D36187	WORD	OK/NG마스타 G8:RR LH "T" REAL Data 차이 <RG3 EV>
D36190	WORD	W500 G9:RR LH "L" REAL Data 차이 <RG3 EV>
D36192	WORD	OK/NG마스타 G9:RR LH "L" REAL Data 차이 <RG3 EV>
D36195	WORD	W500 G10:RR LH "H" REAL Data 차이 <RG3 EV>
D36197	WORD	OK/NG마스타 G10:RR LH "H" REAL Data 차이 <RG3 EV>
D36200	WORD	W500 G11:RR RH "T" REAL Data 차이 <RG3 EV>
D36202	WORD	OK/NG마스타 G11:RR RH "T" REAL Data 차이 <RG3 EV>
D36205	WORD	W500 G12:RR RH "L" REAL Data 차이 <RG3 EV>
D36207	WORD	OK/NG마스타 G12:RR RH "L" REAL Data 차이 <RG3 EV>
D36210	WORD	W500 G13:RR RH "H" REAL Data 차이 <RG3 EV>
D36212	WORD	OK/NG마스타 G13:RR RH "H" REAL Data 차이 <RG3 EV>
D36250	WORD	W600 G1:CTR "L" REAL Data 차이 <RG3 EV>
D36255	WORD	W600 G2:FRT LH "T" REAL Data 차이 <RG3 EV>
D36260	WORD	W600 G3:FRT LH "L" REAL Data 차이 <RG3 EV>
D36265	WORD	W600 G4:FRT LH "H" REAL Data 차이 <RG3 EV>
D36270	WORD	W600 G5:FRT RH "T" REAL Data 차이 <RG3 EV>
D36275	WORD	W600 G6:FRT RH "L" REAL Data 차이 <RG3 EV>
D36280	WORD	W600 G7:FRT RH "H" REAL Data 차이 <RG3 EV>
D36285	WORD	W600 G8:RR LH "T" REAL Data 차이 <RG3 EV>
D36290	WORD	W600 G9:RR LH "L" REAL Data 차이 <RG3 EV>
D36295	WORD	W600 G10:RR LH "H" REAL Data 차이 <RG3 EV>
D36300	WORD	W600 G11:RR RH "T" REAL Data 차이 <RG3 EV>
D36305	WORD	W600 G12:RR RH "L" REAL Data 차이 <RG3 EV>
D36310	WORD	W600 G13:RR RH "H" REAL Data 차이 <RG3 EV>
K01892	BIT	비젼 마스타 기동 W300 배출
D27040	WORD	W350 스케너 Data_LH (W400)
D27540	WORD	W350 스케너 Data_RH (W400)
D27060	WORD	W350 스케너 Data_LH (W400 -> HD2)
D27560	WORD	W350 스케너 Data_RH (W400 -> HD2)
D27080	WORD	W350 스케너 Data_LH (HD2 -> W500)
D27580	WORD	W350 스케너 Data_RH (HD2 -> W500)
D29000	WORD	W500 동도 측정 DATA 아스키 (W500 -> HD2)
D01860	WORD	W500 동도 판정 (HD2 -> W600)
D01960	WORD	W350 3D비젼 체크 (HD2 -> W600)
D24800	WORD	W500 동도 측정 DATA 실수 (HD2 -> NG 대차)
D27160	WORD	W350 스케너 Data_LH (HD2 -> NG 대차)
D27660	WORD	W350 스케너 Data_RH (HD2 -> NG 대차)
D30000	WORD	W500 동도 판정 (HD2 -> W700)
D32000	WORD	W500 동도 측정 DATA 실수 (HD2 -> W700)
D27180	WORD	W350 스케너 Data_LH (HD2 -> W700)
D27680	WORD	W350 스케너 Data_RH (HD2 -> W700)
D30030	WORD	W500 동도 판정 (W700 -> HD2)
D32200	WORD	W500 동도 측정 DATA 실수 (W700 -> HD2)
D33800	WORD	W500 동도 측정 DATA 아스키 (W700 -> HD2)
D30060	WORD	W500 동도 판정 (HD2 -> PLT)
D32400	WORD	W500 동도 측정 DATA 실수 (HD2 -> PLT)
D34000	WORD	W500 동도 측정 DATA 아스키 (HD2 -> PLT)
D27200	WORD	W350 스케너 Data_LH (W700 -> HD2)
D27220	WORD	W350 스케너 Data_LH (HD2 -> PLT)
D27700	WORD	W350 스케너 Data_RH (W700 -> HD2)
D27720	WORD	W350 스케너 Data_RH (HD2 -> PLT)
P0050C	BIT	W10 RH 1차 클램프 잠김1
P0050E	BIT	W10 RH 1차 클램프 잠김2
M10821	BIT	R08 HD2 (In18) PLT-A PLT 사양 확인 
M10824	BIT	R08 HD2 (In21) PLT-B PLT 사양 확인 
K00003	BIT	차종.3 RS4
M10712	BIT	R07 HD1 (In03) 차종3
M10713	BIT	R07 HD1 (In04) 차종4
M10714	BIT	R07 HD1 (In05) 차종5
M10715	BIT	R07 HD1 (In06) 차종6
M10716	BIT	R07 HD1 (In07) 차종7
M10717	BIT	R07 HD1 (In08) 차종8
M10812	BIT	R08 HD2 (In03) 차종3
M10813	BIT	R08 HD2 (In04) 차종4
M10814	BIT	R08 HD2 (In05) 차종5
M10815	BIT	R08 HD2 (In06) 차종6
M10816	BIT	R08 HD2 (In07) 차종7
M10817	BIT	R08 HD2 (In08) 차종8
T0217	BIT/WORD	W10 RH 사양감지 체크완료 지연
M01006	BIT	W250 서보 동작가능
M0100B	BIT	W250 상부 안전센서 정상
M0100C	BIT	W250 하부 안전세서 정상
M0100D	BIT	W250 안전매트 정상
M01060	BIT	W250 원위치복귀 Pb (XP)
M01074	BIT	W250 4차 기동
T1003	BIT/WORD	W250 Air Blow On TMR
T1016	BIT/WORD	W250 파트이상 (누락)지연
T1018	BIT/WORD	W250 서보 위치이상 지연
T1019	BIT/WORD	W250 서보 근접센서 위치이상 Tmr
P0241C	BIT	W70 기동-L
P0241D	BIT	W70 기동-R
P0241E	BIT	W70 원점복귀
D06230	WORD	Label Text.6 Count Data
D00065	WORD	Barcode QR Code Count Data
D00060	WORD	Label Count
D06200	WORD	Label "Year"
D06202	WORD	Label "Month"
D06203	WORD	Label "Day"
D00067	WORD	Barcode QR Code Count ReData
D06210	WORD	Label QR Code Count
D06236	WORD	Label TEXT.6 Count ReData
D06220	WORD	Label TEXT.6 Count Send
D21050	WORD	Label QR Code "0,6,GS,V"
D21054	WORD	Label QR Code "GS,P"
D21060	WORD	Label QR Code "GS,S"
D21068	WORD	Label QR Code "GS,T"
D06201	WORD	Label Year, Month, Day
D21069	WORD	Label QR Code Date Year,Month,Day Send
D21074	WORD	Label QR Code (A0) Send
D21075	WORD	Label QR Code Count Send
D05900	WORD	Lable QR Code Worker Data
D21090	WORD	Label Text.6 Count Send
D20500	WORD	Label QR Code ([)>RS) Send
D20540	WORD	Label Text.5 Date Send
D20541	WORD	Label Text.5 Date Send
D20542	WORD	Label Text.5 Date Send
D20543	WORD	Label Text.5 Date Send
D20544	WORD	Label Text.5 Date Send
D20550	WORD	Label QR Code "0,6,GS,V"
D20554	WORD	Label QR Code "GS,P"
D20560	WORD	Label QR Code "GS,S"
D20563	WORD	Label le QR Code "GS,E"
D20568	WORD	Label QR Code "GS,T"
D20569	WORD	Label QR Code Date Year,Month,Day Send
D20573	WORD	Label QR Code Worker Data
D20574	WORD	Label QR Code (A0) Send
D20575	WORD	Label QR Code Count Send
D20590	WORD	Label Text.6 Count Send
D20541.0	BIT	/
D20541.8	BIT	Label "Month1"
D20542.0	BIT	Label "Month2"
D20542.8	BIT	/
D00099.0	BIT	Label Manual Print
M08511	BIT	ZEBRA Label Head Send
M08512	BIT	ZEBRA Text1 Position Send
M08513	BIT	ZEBRA Text2 Position Send 
M08521	BIT	ZEBRA Text1 Data Send
M08522	BIT	ZEBRA Text2 Data Send
M08523	BIT	ZEBRA Text3 Data Send
M08514	BIT	ZEBRA Text3 Position Send
M08515	BIT	ZEBRA Text4 Position Send
M08524	BIT	ZEBRA Text4 Data Send
M08525	BIT	ZEBRA Text5 Data Send
M08516	BIT	ZEBRA Text5 Position Send
M08517	BIT	ZEBRA Text6 Position Send
M08526	BIT	ZEBRA Text6 Data Send
M08518	BIT	ZEBRA 2D Code Position Send
M08527	BIT	ZEBRA 2D Code Data Send
M08550	BIT	Label Print Complete
P02417	BIT	W70 공기압력
P0241A	BIT	W70 광 안전장치_상부1
P0241B	BIT	W70 광 안전장치_상부2
P02400	BIT	W70 클램프 전진1
P02402	BIT	W70 클램프 전진2
P02404	BIT	W70 클램프 전진3
P02406	BIT	W70 클램프 전진4
P02401	BIT	W70 클램프 후진1
P02403	BIT	W70 클램프 후진2
P02405	BIT	W70 클램프 후진3
P02407	BIT	W70 클램프 후진4
P02408	BIT	W70 동도 유니트 상승1
P0240A	BIT	W70 동도 유니트 상승2
P0240C	BIT	W70 동도 유니트 상승3
P02409	BIT	W70 동도 유니트 하강1
P0240B	BIT	W70 동도 유니트 하강2
P0240D	BIT	W70 동도 유니트 하강3
P02410	BIT	W70 제품확인1
P02411	BIT	W70 제품확인2
P02420	BIT	W70 클램프 잠김 Sol
P02421	BIT	W70 클램프 풀림 Sol
P02422	BIT	W70 동도 유니트 상승 Sol
P02423	BIT	W70 동도 유니트 하강 Sol
P02440	BIT	[From] W500 TOE/CAM Ready
P02441	BIT	[From] W500 TOE/CAM ERROR
P02442	BIT	[From] W500 TOE/CAM N.G
P02443	BIT	[From] W500 TOE/CAM O.K
P02450	BIT	[To Dongdo] W500TOE/CAM Model1
P02451	BIT	[To Dongdo] W500TOE/CAM Model2
P02452	BIT	[To Dongdo] W500TOE/CAM Model4
P02453	BIT	[To Dongdo] W500TOE/CAM Model8
P02454	BIT	[To Dongdo] W500 TOE/CAM Check Start
D41000	WORD	W70 동도 버퍼
D44000	WORD	W70 동도 측정 DATA
D41003	WORD	P1 ASCII Data
D41008	WORD	P2 ASCII Data
D41013	WORD	P3 ASCII Data
D41018	WORD	P4 ASCII Data
D41023	WORD	P5 ASCII Data
D41028	WORD	P6 ASCII Data
D41033	WORD	P7 ASCII Data
D42000	WORD	동도 읽을 위치 1
D42001	WORD	동도 읽을 자릿수 1
D42002	WORD	동도 읽을 위치 2
D42003	WORD	동도 읽을 자릿수 2
D42010	WORD	P1 ASCII Data
D42020	WORD	P2 ASCII Data
D42030	WORD	P3 ASCII Data
D42040	WORD	P4 ASCII Data
D42050	WORD	P5 ASCII Data
D42060	WORD	P6 ASCII Data
D42070	WORD	P7 ASCII Data
D44010	WORD	P1 REAL Data
D44020	WORD	P2 REAL Data
D44030	WORD	P3 REAL Data
D44040	WORD	P4 REAL Data
D44050	WORD	P5 REAL Data
D44060	WORD	P6 REAL Data
D44070	WORD	P7 REAL Data
D45007	WORD	Data 절대 상/하한치
D45010	WORD	P1 REAL Data 하한치
D45012	WORD	P1 REAL Data 하한치 절대
D45015	WORD	P1 REAL Data 상한치
D45017	WORD	P1 REAL Data 상한치 절대
D45020	WORD	P2 REAL Data 하한치
D45022	WORD	P2 REAL Data 하한치 절대
D45025	WORD	P2 REAL Data 상한치
D45027	WORD	P2 REAL Data 상한치 절대
D45030	WORD	P3 REAL Data 하한치
D45032	WORD	P3 REAL Data 하한치 절대
D45035	WORD	P3 REAL Data 상한치
D45037	WORD	P3 REAL Data 상한치 절대
D45040	WORD	P4 REAL Data 하한치
D45042	WORD	P4 REAL Data 하한치 절대
D45045	WORD	P4 REAL Data 상한치
D45047	WORD	P4 REAL Data 상한치 절대
D45050	WORD	P5 REAL Data 하한치
D45052	WORD	P5 REAL Data 하한치 절대
D45055	WORD	P5 REAL Data 상한치
D45057	WORD	P5 REAL Data 상한치 절대
D45060	WORD	P6 REAL Data 하한치
D45062	WORD	P6 REAL Data 하한치 절대
D45065	WORD	P6 REAL Data 상한치
D45067	WORD	P6 REAL Data 상한치 절대
D45070	WORD	P7 REAL Data 하한치
D45072	WORD	P7 REAL Data 하한치 절대
D45075	WORD	P7 REAL Data 상한치
D45077	WORD	P7 REAL Data 상한치 절대
D46010	WORD	P1 REAL 스펙Data 
D46012	WORD	P1 REAL 하한치
D46017	WORD	P1 REAL 상한치
D46020	WORD	P2 REAL 스펙Data 
D46030	WORD	P3 REAL 스펙Data 
D46040	WORD	P4 REAL 스펙Data 
D46042	WORD	P4 REAL 하한치
D46047	WORD	P4 REAL 상한치
D46050	WORD	P5 REAL 스펙Data 
D46052	WORD	P5 REAL 하한치
D46057	WORD	P5 REAL 상한치
D46060	WORD	P6 REAL 스펙Data 
D46062	WORD	P6 REAL 하한치
D46067	WORD	P6 REAL 상한치
D46070	WORD	P7 REAL 스펙Data 
D46072	WORD	P7 REAL 하한치
D46077	WORD	P7 REAL 상한치
D46150	WORD	P1 REAL Data 차이
D46155	WORD	P2 REAL Data 차이
D46160	WORD	P3 REAL Data 차이
D46165	WORD	P4 REAL Data 차이
D46170	WORD	P5 REAL Data 차이
D46175	WORD	P6 REAL Data 차이
D46180	WORD	P7 REAL Data 차이
D11007	WORD	W70 Scan Data 1
D11009	WORD	W70 Scan Data 3
D11011	WORD	W70 Scan Data 5
D31400	WORD	PLC->PC W70 스케너 Data
D31500	WORD	PLC->PC W70 동도 측정 Data
D00059.0	BIT	1 Shift Time
D00059.1	BIT	2 Shift Time
D14103.3	BIT	W70 Check OK
D14103.4	BIT	W70 Check NG
D14103.5	BIT	W70 Scan Comple
D14101.5	BIT	W70 Scan Compl
D14103.E	BIT	W70 Loading
D14101.E	BIT	W70 Loading Check
D20576	WORD	Barcord Print Data1
D15002.9	BIT	W70 수동모드
P02428	BIT	W70 타워램프-R
P02429	BIT	W70 타워램프-G
D43010	WORD	W70 P1 REAL Data_Master
D43020	WORD	W70 P2 REAL Data_Master
D43030	WORD	W70 P3 REAL Data_Master
D43040	WORD	W70 P4 REAL Data_Master
D43050	WORD	W70 P5 REAL Data_Master
D43060	WORD	W70 P6 REAL Data_Master
D43070	WORD	W70 P7 REAL Data_Master
D48150	WORD	W70 P1 REAL Data 차이 _Master
D48155	WORD	W70 P2 REAL Data 차이 _Master
D48160	WORD	W70 P3 REAL Data 차이 _Master
D48165	WORD	W70 P4 REAL Data 차이 _Master
D48170	WORD	W70 P5 REAL Data 차이 _Master
D48175	WORD	W70 P6 REAL Data 차이 _Master
D48180	WORD	W70 P7 REAL Data 차이 _Master
K01780	BIT	W70 OK 마스타 선택중
K01781	BIT	W70 OK 마스타 체크 기동
M03981	BIT	W70 OK 마스타 체크 Off T/K
M03980	BIT	W70 OK 마스타 체크 On T/K
M03984	BIT	W70 OK 마스타 예약기동
K01990	BIT	W70 OK 마스타 선택중
M05960	BIT	W70 OK 마스타 체크 On T/K
M05964	BIT	W70 OK 마스타 예약기동
K01991	BIT	W70 OK 마스타 체크 기동
M05961	BIT	W70 OK 마스타 체크 Off T/K
M05970	BIT	W70 OK 마스타 Start Lamp
R02600	WORD	W70 OK 마스타체크 최종점검 일자 년
M05971	BIT	W70 OK 마스타 주간 초품 확인시간
M05972	BIT	W70 OK 마스타 주간 중품 확인시간
M05973	BIT	W70 OK 마스타 야간 초품 확인시간
M05974	BIT	W70 OK 마스타 야간 중품 확인시간
M05951	BIT	W70 OK 마스타 주간 초품 체크 완료
M05952	BIT	W70 OK 마스타 주간 중품 체크 완료
M05953	BIT	W70 OK 마스타 야간 초품 체크 완료
M05954	BIT	W70 OK 마스타 야간 중품 체크 완료
D00029	WORD	W70 OK 마스타운영 시간설정 비번
D05822	WORD	W70 OK 마스타 주간 초품 시작 시간
D05823	WORD	W70 OK 마스타 주간 초품 끝 시간
D05824	WORD	W70 OK 마스타 주간 중품 시작 시간
D05825	WORD	W70 OK 마스타 주간 중품 끝 시간
D05826	WORD	W70 OK 마스타 야간 초품 시작 시간
D05828	WORD	W70 OK 마스타 야간 중품 시작 시간
D05827	WORD	W70 OK 마스타 야간 초품 끝 시간
D05829	WORD	W70 OK 마스타 야간 중품 끝 시간
D05840	WORD	W70 OK 마스타 주간 초품 정보
D05841	WORD	W70 OK 마스타 주간 중품 정보
D05842	WORD	W70 OK 마스타 야간 초품 정보
D05843	WORD	W70 OK 마스타 야간 중품 정보
D05820	WORD	W70 OK 마스타 확인 정보 클리어 시
D05821	WORD	W70 OK 마스타 확인 정보 클리어 분
M0597A	BIT	W70 OK마스타 주간 초품 체크 지령
M0597B	BIT	W70 OK 마스타 주간 중품 체크 지령
M0597C	BIT	W70 OK 마스타 야간 초품 체크 지령
M0597D	BIT	W70 OK 마스타 야간 중품 체크 지령
P11100	BIT	R11 HD3 Running
P11101	BIT	R11 HD3 Servo_ON
P11103	BIT	R11 HD3 Error
P11105	BIT	R11 HD3 REMOTE Mode
P11106	BIT	R11 HD3 PLAY Mode
P11107	BIT	R11 HD3 TEACH 모드
P1110A	BIT	R11 HD3 HOME Position
P11110	BIT	R11 HD3 (Ot01) W50 간섭무
P11111	BIT	R11 HD3 (Ot02) W60-1 간섭무
P11112	BIT	R11 HD3 (Ot03) W60-2 간섭무
P11113	BIT	R11 HD3 (Ot03) W60-3 간섭무
P11114	BIT	R11 HD3 (Ot05) W70 간섭무
P11115	BIT	R11 HD3 (Ot06)
P11116	BIT	R11 HD3 (Ot07)
P11117	BIT	R11 HD3 (Ot08)
P11118	BIT	R11 HD3 (Ot09) W50 언로딩 완료
P11119	BIT	R11 HD3 (Ot09)
P1111A	BIT	R11 HD3 (Ot11) W60-1 로딩 완료
P1111B	BIT	R11 HD3 (Ot12) W60-1 언로딩 완료
P1111C	BIT	R11 HD3 (Ot13) W60-2 로딩 완료
P1111D	BIT	R11 HD3 (Ot14) W60-1 언로딩 완료
P1111E	BIT	R11 HD3 (Ot15) W60-3 로딩 완료
P1111F	BIT	R11 HD3 (Ot16) W60-1 언로딩 완료
P11120	BIT	R11 HD3 (Ot17) W70 로딩완료
P11121	BIT	R11 HD3 (Ot18)
P11122	BIT	R11 HD3 (Ot19)
P11123	BIT	R11 HD3 (Ot20)
P11124	BIT	R11 HD3 (Ot21)
P11125	BIT	R11 HD3 (Ot22)
P11126	BIT	R11 HD3 (Ot23)
P11127	BIT	R11 HD3 (Ot24)
P11128	BIT	R11 HD3 (Ot25)
P11129	BIT	R11 HD3 (Ot26) R11 HD3->R01 인터록
P1112A	BIT	R11 HD3 (Ot27)
P1112B	BIT	R11 HD3 (Ot28)
P1112C	BIT	R11 HD3 (Ot29)
P1112D	BIT	R11 HD3 (Ot30)
P1112F	BIT	R11 HD3 (Ot32) 비상정지
P11131	BIT	R11 HD4 (Ot34)
P11132	BIT	R11 HD3 (Ot35)
P11133	BIT	R11 HD3 (Ot36)
P11134	BIT	R11 HD3 (Ot37)
P11135	BIT	R11 HD3 (Ot38)
P11136	BIT	R11 HD3 (Ot39)
P11137	BIT	R11 HD3 (Ot40)
P11141	BIT	R11 HD3 (Ot50) 그리퍼1 클램프 잠김요구
P11142	BIT	R11 HD3 (Ot51) 그리퍼1 클램프 풀림요구
P11143	BIT	R11 HD3 (Ot52) 그리퍼1 핀 전진요구
P11144	BIT	R11 HD3 (Ot53) 그리퍼1 핀 후진요구
P11145	BIT	R11 HD3 (Ot54)
P11146	BIT	R11 HD3 (Ot55) 그리퍼2 클램프 잠김요구
P11147	BIT	R11 HD3 (Ot56) 그리퍼2 클램프 풀림요구
P11148	BIT	R11 HD3 (Ot57) 그리퍼2 핀 전진요구
P11149	BIT	R11 HD3 (Ot58)
P1114A	BIT	R11 HD3 (Ot59)
P1114B	BIT	R11 HD3 (Ot60)
P1114C	BIT	R11 HD3 (Ot61)
P1114D	BIT	R11 HD3 (Ot62)
P1114E	BIT	R11 HD3 (Ot63)
P1114F	BIT	R11 HD3 (Ot64)
P11150	BIT	R11 HD3 (Ot65)
P11151	BIT	R11 HD3 (Ot66)
P11152	BIT	R11 HD3 (Ot67)
P11153	BIT	R11 HD3 (Ot68)
P11154	BIT	R11 HD3 (Ot69)
P11155	BIT	R11 HD3 (Ot70)
P11156	BIT	R11 HD3 (Ot71)
P11157	BIT	R11 HD3 (Ot72)
P11158	BIT	R11 HD3 (Ot73)
P11159	BIT	R11 HD3 (Ot74)
P1115A	BIT	R11 HD3 (Ot75)
P1115B	BIT	R11 HD3 (Ot76)
P1115C	BIT	R11 HD3 (Ot77)
P1115D	BIT	R11 HD3 (Ot78)
P1115E	BIT	R11 HD3 (Ot79)
P1115F	BIT	R11 HD3 (Ot80)
P11160	BIT	R11 HD3 (Ot81)
P11161	BIT	R11 HD3 (Ot82)
P11162	BIT	R11 HD3 (Ot83)
P11163	BIT	R11 HD3 (Ot84)
P11164	BIT	R11 HD3 (Ot85)
P11165	BIT	R11 HD3 (Ot86)
P11166	BIT	R11 HD3 (Ot87)
P11167	BIT	R11 HD3 (Ot88)
P11168	BIT	R11 HD3 (Ot89)
P11169	BIT	R11 HD3 (Ot90)
P1116A	BIT	R11 HD3 (Ot91)
P1116B	BIT	R11 HD3 (Ot92)
P1116C	BIT	R11 HD3 (Ot93)
P1116D	BIT	R11 HD3 (Ot94)
P1116E	BIT	R11 HD3 (Ot95)
P1116F	BIT	R11 HD3 (Ot96)
P11170	BIT	R11 HD3 그리퍼 파트감지
P11171	BIT	R11 HD3 그리퍼 핀 후진1
P11172	BIT	R11 HD3 그리퍼 핀 전진1
P11173	BIT	R11 HD3 그리퍼 핀 후진2
P11174	BIT	R11 HD3 그리퍼 핀 전진2
P11175	BIT	R11 HD3 그리퍼 클램프 잠김1
P11176	BIT	R11 HD3 그리퍼 클램프 풀림1
P11177	BIT	R11 HD3 그리퍼 클램프 잠김2
P11178	BIT	R11 HD3 그리퍼 클램프 풀림2
P11179	BIT	R11 HD3 그리퍼 클램프 잠김3
P1117A	BIT	R11 HD3 그리퍼 클램프 풀림3
P1117B	BIT	R11 HD3 그리퍼1 No.2 너트감지 파트1
P1117C	BIT	R11 HD3 그리퍼1 No.2 너트감지 파트2
P1117D	BIT	R11 HD3 그리퍼1 클램프 잠김2
P1117E	BIT	R11 HD3 그리퍼1 클램프 풀림2
P1118E	BIT	HD-2 H/D Robot Air Press S/W
M11100	BIT	R11 HD3 External RUN
M11101	BIT	R11 HD3 Servo_ON
M11103	BIT	R11 HD3 Error Reset
M11105	BIT	R11 HD3 REMInE Selet
M11106	BIT	R11 HD3 PLAY Select
M11107	BIT	R11 HD3 TEACH Select
M1110A	BIT	OP2 RobIn WELD ON
M11110	BIT	R11 HD3 (In01) 차종1
M11111	BIT	R11 HD3 (In02) 차종2
M11112	BIT	R11 HD3 (In03) 차종3
M11113	BIT	R11 HD3 (In04) 차종4
M11114	BIT	R11 HD3 (In05) 차종5
M11115	BIT	R11 HD3 (In06) 차종6
M11116	BIT	R11 HD3 (In07) 차종7
M11117	BIT	R11 HD3 (In08) 차종8
M11118	BIT	R11 HD3 (In09) W50 언로딩 가능
M11119	BIT	R11 HD3 (In10)
M1111A	BIT	R11 HD3 (In11) W60-1 로딩 가능
M1111B	BIT	R11 HD3 (In12) W60-1 언로딩 가능
M1111C	BIT	R11 HD3 (In13) W60-2 로딩 가능
M1111D	BIT	R11 HD3 (In14) W60-2 언로딩 가능
M1111E	BIT	R11 HD3 (In15) W60-3 로딩 가능
M1111F	BIT	R11 HD3 (In16) W60-3 언로딩 가능
M11120	BIT	R11 HD3 (In17) W70 로딩 가능
M11122	BIT	R11 HD3 (In19)
M11124	BIT	R11 HD3 (In21)
M11125	BIT	R11 HD3 (In22)
M11126	BIT	R11 HD3 (In23) W60 FULL
M11127	BIT	R11 HD3 (In24) 강제배출 가능
M11128	BIT	R11 HD3 (In25)
M11129	BIT	R11 HD3 (In26) R11 HD3<-R01 인터록
M1112A	BIT	R11 HD3 (In27)
M1112B	BIT	R11 HD3 (In28)
M1112C	BIT	R11 HD3 (In29)
M1112D	BIT	R11 HD3 (In30)
M1112E	BIT	R11 HD3 (In31) 외부 비상정지
M1112F	BIT	R11 HD3 (In32) 외부 일시정지
M11131	BIT	R11 HD3 (In34)
M11132	BIT	R11 HD3 (In35)
M11133	BIT	R11 HD3 (In36)
M11134	BIT	R11 HD3 (In37)
M11135	BIT	R11 HD3 (In38)
M11136	BIT	R11 HD3 (In39)
M11137	BIT	R11 HD3 (In40)
M11142	BIT	R11 HD3 (In51) 그리퍼1 클램프 풀림
M11143	BIT	R11 HD3 (In52) 그리퍼1 핀 전진
M11144	BIT	R11 HD3 (In53) 그리퍼1 핀 후진
M11145	BIT	R11 HD3 (In54) 그리퍼2 파트감지
M11148	BIT	R11 HD3 (In57) 그리퍼2 핀 전진
M11149	BIT	R11 HD3 (In58) 그리퍼2 핀 후진
M1114A	BIT	R11 HD3 (In59)
M1114B	BIT	R11 HD3 (In60)
M1114C	BIT	R11 HD3 (In61)
M1114D	BIT	R11 HD3 (In62)
M1114E	BIT	R11 HD3 (In63)
M1114F	BIT	R11 HD3 (In64)
M11150	BIT	R11 HD3 (In65)
M11151	BIT	R11 HD3 (In66)
M11152	BIT	R11 HD3 (In67)
M11153	BIT	R11 HD3 (In68)
M11154	BIT	R11 HD3 (In69)
M11155	BIT	R11 HD3 (In70)
M11156	BIT	R11 HD3 (In71)
M11157	BIT	R11 HD3 (In72)
M11158	BIT	R11 HD3 (In73)
M11159	BIT	R11 HD3 (In74)
M1115A	BIT	R11 HD3 (In75)
M1115B	BIT	R11 HD3 (In76)
M1115C	BIT	R11 HD3 (In77)
M1115D	BIT	R11 HD3 (In78)
M1115E	BIT	R11 HD3 (In79)
M1115F	BIT	R11 HD3 (In80)
M11160	BIT	R11 HD3 (In81)
M11161	BIT	R11 HD3 (In82)
M11162	BIT	R11 HD3 (In83)
M11163	BIT	R11 HD3 (In84)
M11164	BIT	R11 HD3 (In85)
M11165	BIT	R11 HD3 (In86)
M11166	BIT	R11 HD3 (In87)
M11167	BIT	R11 HD3 (In88)
M11168	BIT	R11 HD3 (In89)
M11169	BIT	R11 HD3 (In90)
M1116A	BIT	R11 HD3 (In91)
M1116B	BIT	R11 HD3 (In92)
M1116C	BIT	R11 HD3 (In93)
M1116D	BIT	R11 HD3 (In94)
M1116E	BIT	R11 HD3 (In95)
M1116F	BIT	R11 HD3 (In96)
M11170	BIT	R11 HD3 그리퍼2 핀 전진 SOL
M11171	BIT	R11 HD3 그리퍼2 핀 후진 SOL
M11172	BIT	R11 HD3 그리퍼2 클램프 잠김 SOL
M11173	BIT	R11 HD3 그리퍼2 클램프 풀림 SOL
M11174	BIT	R11 HD3 그리퍼1 핀 전진 Sol
M11175	BIT	R11 HD3 그리퍼1 핀 후진 Sol
M11176	BIT	R11 HD3 그리퍼1 클램프 잠김 Sol
M11177	BIT	R11 HD3 그리퍼1 클램프 풀림 Sol
M11190	BIT	R11 HD3 그리퍼 파트감지 없음
M11146	BIT	R11 HD3 (In55) 그리퍼2 클램프 잠김
M11147	BIT	R11 HD3 (In56) 그리퍼2 클램프 풀림
P1112E	BIT	R11 HD3 (Ot31)
P02414	BIT	W60-1 제품확인
P02413	BIT	W60-2 제품확인
P02412	BIT	W60-3 제품확인
M0107A	BIT	W250 2차 작업준비
M16289	BIT	OP1 R11 Seleted
P10129	BIT	R01 (OT26)
M16520	BIT	로워판넬 라인 강제배출 Mode on
P11130	BIT	R11 HD3 (Ot33) W50 툴핀 하강요구
M11130	BIT	R11 HD3 (In33) W50 툴핀 하강완료
P11140	BIT	R11 HD3 (Ot49)
P11138	BIT	R11 HD3 (Ot41)
P11139	BIT	R11 HD3 (Ot42)
P1113A	BIT	R11 HD3 (Ot43)
P1113B	BIT	R11 HD3 (Ot44)
P1113C	BIT	R11 HD3 (Ot45)
P1113D	BIT	R11 HD3 (Ot46)
P1113E	BIT	R11 HD3 (Ot47)
P1113F	BIT	R11 HD3 (Ot48)
M11140	BIT	R11 HD3 (In49) 그리퍼1 파트감지
M11141	BIT	R11 HD3 (In50) 그리퍼1 클램프 잠김
M11138	BIT	R11 HD3 (In41)
M11139	BIT	R11 HD3 (In42)
M1113A	BIT	R11 HD3 (In43)
M1113B	BIT	R11 HD3 (In44)
M1113C	BIT	R11 HD3 (In45)
M1113E	BIT	R11 HD3 (In47)
M1113D	BIT	R11 HD3 (In46)
M1113F	BIT	R11 HD3 (In48)
M0007E	BIT	OP1 Robot11 Gripper Error
M0007F	BIT	OP1 Robot11 Part Error
M16269	BIT	OP1 R11 Select Pb
D15002.A	BIT	W70 구형판넬 사용
D15002.B	BIT	W50 언로딩모드 작업자
P02424	BIT	W70 P1 측정 OK LAMP
P02425	BIT	W70 P1 측정 NG LAMP
P02426	BIT	W70 P2 측정 OK LAMP
P02427	BIT	W70 P2 측정 NG LAMP
P0242B	BIT	W70 P3 측정 OK LAMP
P0242C	BIT	W70 P3 측정 NG LAMP
P02456	BIT	W70 P4 측정 OK LAMP
P02457	BIT	W70 P4 측정 NG LAMP
P02458	BIT	W70 P5 측정 OK LAMP
P02459	BIT	W70 P5 측정 NG LAMP
P0245A	BIT	W70 P6 측정 OK LAMP
P0245B	BIT	W70 P6 측정 NG LAMP
P0245C	BIT	W70 P7 측정 OK LAMP
P0245D	BIT	W70 P7 측정 NG LAMP
P0245E	BIT	W70 동도 측정 O.K LAMP
P0245F	BIT	W70 동도 측정 N.G LAMP
D15507	WORD	OP1 터치 현재선택
D15508	WORD	OP1 현재 차종 정보
D15509	WORD	OP1 현재 차종 정보
D15514	WORD	Car Type Exchange Possible State
M16530	BIT	로워판넬 Line 강제배출 Mode On
T0009	BIT/WORD	Line 강제배출 Mode On Delay Tmr
M16521	BIT	로워판넬 Line 강제배출 Mode Off Pb
T0017	BIT/WORD	Line 강제배출 Mode Off Delay Tmr
D18701	WORD	W50 차종 정보
D18702	WORD	W50 -> W60 HD3 버퍼
D18703	WORD	W60-1 차종 정보
D18704	WORD	W60-2 차종 정보
D18705	WORD	W60-3 차종 정보
D18706	WORD	W60 -> W70 HD3 버퍼
D18707	WORD	W70 차종정보
D46022	WORD	RG3 하한치
D46027	WORD	RG3 상한치
D46032	WORD	RS4 하한치
D46037	WORD	RS4 상한치
K00011	BIT	로워판넬 라인 차종.1 RG3
K00012	BIT	로워판넬 라인 차종.2 RG3 EV
M11121	BIT	R11 HD3 (In18) W70 언로딩 가능
M11123	BIT	R11 HD3 (In20) 마스터 언로딩 가능
P1061B	BIT	R06 (OT12)
D14102.5	BIT	Car Type-1(LWR PNL)
D14102.6	BIT	Car Type-2(LWR PNL)
D14103.F	BIT	Master Check Mode (LWR PNL)
M0006A	BIT	Car Type Change Request
M0006B	BIT	Car Type Change Start
T0092	BIT/WORD	Car Type Change End
T0093	BIT/WORD	Car Type Change Signal Reset
D20577	WORD	Barcord Print Data1-1
D20558	WORD	Barcord Print Data1
K00121	BIT	RG3 EV 푸셔 작업 완료
D00160	WORD	W50 RG3 EV 푸셔 상승완료 지연설정
P00312	BIT	W10 LH 1차 클램프 잠김4
P00313	BIT	W10 LH 1차 클램프 풀림4
P1110E	BIT	R11 H/D3 비상정지
D15002.C	BIT	W50 푸셔 바이패스 ON
K05000	BIT	W350 RH 바코드 스켄 OK test
K00013	BIT	로워판넬 라인 차종.3 RG3/RS4
T0081	BIT/WORD	W50 상부광센스
K00031	BIT	W50 작업자 라인 진입
K00041	BIT	W50  광센서 상.하부 동시 이상
T0082	BIT/WORD	W70 상부광센스
K00032	BIT	W70 작업자 라인 진입
K00042	BIT	W70  광센서 상.하부 동시 이상
D00131	WORD	W50 작업자  안전확보  데이트 이상
D00132	WORD	W70 작업자  안전확보  데이트 이상
D00133	WORD	W100 작업자  안전확보  데이트 이상
T0083	BIT/WORD	W100 상부광센스
K00033	BIT	W100 작업자 라인 진입
K00043	BIT	W100  광센서 상.하부 동시 이상
D00134	WORD	W600 작업자  안전확보  데이트 이상
T0084	BIT/WORD	W600 상부광센스
K00044	BIT	W600  광센서 상.하부 동시 이상
K00034	BIT	W600 작업자 라인 진입
T0086	BIT/WORD	W50공정 상.하부 동시감지 시간지연
T0087	BIT/WORD	W70공정 상.하부 동시감지 시간지연
T0088	BIT/WORD	W100공정 상.하부 동시감지 시간지연
T0089	BIT/WORD	W600공정 상.하부 동시감지 시간지연
K00004	BIT	차종.4 HDP
K00014	BIT	로워 판넬 차종4 RS4 HDP
T8001	BIT/WORD	상부 광센스 지연
M07001	BIT	트리거 온
R05001.1	BIT	클리어 비트
R05000.1	BIT	카메라 촬영 시작
R04000.1	BIT	카메라 촬영 완료
R04000.0	BIT	카메라 준비 완료
R05000.0	BIT	카메라 촬영 준비
R05004	WORD	카메라 차종
R05005	WORD	카메라 쵤영 위치
M10646	BIT	R06 (IN55)
M10644	BIT	R06 (IN53)
M10647	BIT	R06 (IN56)
R05005.0	BIT	촬영 위치 Bit
P10647	BIT	R06 (OT56)
T3002	BIT/WORD	카메라 촬영 시작 유지시간
T3001	BIT/WORD	카메라 촬영 완료 차단시간
K00050	BIT	카메라 촬영 완료
P10648	BIT	R06 (OT57)
D28005	WORD	스캐너 카운터
D08000	WORD	스케너Data
D06041	WORD	W200 R05 용접누락 판정결과 (EV)
D06042	WORD	W200 R05 용접누락 판정결과 (RS4)
D06031	WORD	W200 R04 용접누락 판정결과 (EV)
D06032	WORD	W200 R04 용접누락 판정결과 (RS4)
D06021	WORD	W100 R03 용접누락 판정결과 [EV]
D06022	WORD	W100 R03 용접누락 판정결과 [RS4]
D06011	WORD	W100 R02 용접누락 판정결과 [EV]
D06012	WORD	W100 R02 용접누락 판정결과 [RS4]
D06001	WORD	W50 R01 용접누락 판정결과 [EV]
D06002	WORD	W50 R01 용접누락 판정결과 [RS4]
D08385	WORD	R05 표준시간 최소 용접시간 설정[EV]
D08386	WORD	R05 표준시간 최대 용접시간 [EV]
D08387	WORD	W200 R05 용접구간 카운터[EV]
D08388	WORD	W200 R05 용접구간 카운터설정[EV]
D08390	WORD	R05 표준시간 최소 용접시간 설정[RS4]
D08391	WORD	R05 표준시간 최대 용접시간 [RS4]
D08392	WORD	W200 R05 용접구간 카운터[RS4]
D08393	WORD	W200 R05 용접구간 카운터설정[RS4]
D08365	WORD	R04 표준시간 최소 용접시간 설정[EV]
D08366	WORD	R04 표준시간 최대 용접시간 [EV]
D08367	WORD	W200 R04 용접구간 카운터[EV]
D08368	WORD	W200 R04 용접구간 카운터설정[EV]
D08370	WORD	R04 표준시간 최소 용접시간 설정[RS4]
D08371	WORD	R04 표준시간 최대 용접시간 [RS4]
D08372	WORD	W200 R04 용접구간 카운터[RS4]
D08373	WORD	W200 R04 용접구간 카운터설정[RS4]
D08345	WORD	R03 표준시간 최소 용접시간 설정[EV]
D08346	WORD	R03 표준시간 최대 용접시간 [EV]
D08347	WORD	W100 R03 용접구간 카운터[EV]
D08348	WORD	W100 R03 용접구간 카운터설정[EV]
D08350	WORD	R03 표준시간 최소 용접시간 설정[RS4]
D08351	WORD	R03 표준시간 최대 용접시간 [RS4]
D08352	WORD	W100 R03 용접구간 카운터[RS4]
D08353	WORD	W100 R03 용접구간 카운터설정[RS4]
D08325	WORD	R02 표준시간 최소 용접시간 설정[EV]
D08326	WORD	R02 표준시간 최대 용접시간  [EV]
D08327	WORD	W100 R02 용접구간 카운터[EV]
D08328	WORD	W100 R02 용접구간 카운터설정[EV]
D08330	WORD	R02 표준시간 최소 용접시간 설정[RS4]
D08331	WORD	R02 표준시간 최대 용접시간  [RS4]
D08332	WORD	W100 R02 용접구간 카운터  [RS4]
D08333	WORD	W100 R02 용접구간 카운터설정[RS4]
D08305	WORD	R01 표준시간 최소 용접시간 설정 [EV]
D08306	WORD	R01 표준시간 최대 용접시간 [EV]
D08307	WORD	W50 R01 용접구간 카운터
D08308	WORD	W50 R01 용접구간 카운터설정 [EV]
D08310	WORD	R01 표준시간 최소 용접시간 설정 [RS4]
D08311	WORD	R01 표준시간 최대 용접시간 [RS4]
D08312	WORD	W50 R01 용접구간 카운터
D08313	WORD	W50 R01 용접구간 카운터설정 [RS4]
D18048.1	BIT	R05 용접누락 이상 [RS4]
D18037.1	BIT	R04 용접누락 이상 [EV]
D18038.1	BIT	R04 용접누락 이상 [RS4]
D18027.1	BIT	R03 용접누락 이상 [EV]
D18028.1	BIT	R03 용접누락 이상 [RS4]
D18017.1	BIT	R02 용접누락 이상 [EV]
D18018.1	BIT	R02 용접누락 이상 [RS4]
D18007.1	BIT	R01 용접누락 이상 [EV]
D18008.1	BIT	R01 용접누락 이상 [RS4]
D18048.2	BIT	R05 구간누락 이상 [RS4]
D18048.3	BIT	R05 용접시간/구간누락 이상 [RS4]
D18047.2	BIT	R05 구간누락 이상 [EV]
D18047.3	BIT	R05 용접시간/구간누락 이상 [EV]
D18046.2	BIT	R05 구간누락 이상 [RG3]
D18046.3	BIT	R05 용접시간/구간누락 이상 [RG3]
D18047	WORD	R05 용접누락 이상 [EV]
D18046	WORD	R05 용접누락 이상 [RG3]
D18047.1	BIT	R05 용접누락 이상 [EV]
M10728	BIT	R07 HD1 (In25) R07 HD1<-R6 인터록 (바코드)
P10727	BIT	R07 HD1 (Ot24) HD1->R6 인터록
P10726	BIT	R07 비전1차 촬영위치 도착 HD1 (Ot23)
M10726	BIT	R07 HD1 (In23) 비전1차 촬영완료
M10090	BIT	카메라 촬영완료
P10626	BIT	R06 (OT23)
P0241F	BIT	W70 비상정지 PB
D70013	WORD	시
D70014	WORD	분
D70015	WORD	초
D70016	WORD	요일
D70035	WORD	Item 5 production
D70036	WORD	Item 6 production
D71002	WORD	공파레트 "A" 진입 대기 <--AMR
D71003	WORD	공파레트 "A" 진입중 <--AMR
D71012	WORD	배출 "A" 진입 대기 <--AMR
D71013	WORD	배출 "A" 진입중 <--AMR
D71014	WORD	배출 "A" 완료 <--AMR
D71022	WORD	공파레트 "B" 진입 대기 <--AMR
D71023	WORD	공파레트 "B" 진입중 <--AMR
D71032	WORD	배출 "B" 진입 대기 <--AMR
D71033	WORD	배출 "B" 진입중 <--AMR
D71034	WORD	배출 "B" 완료 <--AMR
D70500	WORD	시간 저장
D70480	WORD	현재 시간
P0031B	BIT	W10 LH 3차 클램프 풀림3
P00518	BIT	W10 RH 3차 클램프 잠김2
P00519	BIT	W10 RH 3차 클램프 풀림2
P00906	BIT	W100 LH 클램프 잠김1
P00907	BIT	W100 LH 클램프 풀림1
P00908	BIT	W100 LH 클램프 잠김2
P00909	BIT	W100 LH 클램프 풀림2
P0090A	BIT	W100 LH 클램프 잠김3
P0090B	BIT	W100 LH 클램프 풀림3
P0090C	BIT	W100 LH 클램프 잠김4
P0090D	BIT	W100 LH 클램프 풀림4
P0090E	BIT	W100 LH 클램프 잠김5
P0090F	BIT	W100 LH 클램프 풀림5
P00918	BIT	W100 RH 클램프 잠김1
P00919	BIT	W100 RH 클램프 풀림1
P0091A	BIT	W100 RH 클램프 잠김2
P0091B	BIT	W100 RH 클램프 풀림2
P0091C	BIT	W100 RH 클램프 잠김3
P0091D	BIT	W100 RH 클램프 풀림3
P0091E	BIT	W100 RH 클램프 잠김4
P0091F	BIT	W100 RH 클램프 풀림4
P00920	BIT	W100 RH 클램프 잠김5
P00921	BIT	W100 RH 클램프 풀림5
P00924	BIT	W100 NO.1 클램프 잠김
P00925	BIT	W100 NO.1 클램프 풀림
P00926	BIT	W100 NO.2 클램프 잠김
P00927	BIT	W100 NO.2 클램프 풀림
P01206	BIT	W200 LH 클램프 잠김1
P01207	BIT	W200 LH 클램프 풀림1
P01208	BIT	W200 LH 클램프 잠김2
P01209	BIT	W200 LH 클램프 풀림2
P0120A	BIT	W200 LH 클램프 잠김3
P0120B	BIT	W200 LH 클램프 풀림3
P0120C	BIT	W200 LH 클램프 잠김4
P0120D	BIT	W200 LH 클램프 풀림4
P01214	BIT	W200 RH 클램프 잠김1
P01215	BIT	W200 RH 클램프 풀림1
P01216	BIT	W200 RH 클램프 잠김2
P01217	BIT	W200 RH 클램프 풀림2
P01218	BIT	W200 RH 클램프 잠김3
P01219	BIT	W200 RH 클램프 풀림3
P0121A	BIT	W200 RH 클램프 잠김4
P0121B	BIT	W200 RH 클램프 풀림4
P0152E	BIT	W400 파트확인 [PL]
P1218E	BIT	R21 H/D1 공압 S/W
P1247B	BIT	R24 H/D4 그리퍼1 클램프 풀림4
P1247C	BIT	R24 H/D4 그리퍼1 파트
T0216	BIT/WORD	W10 RH 파트이상 (누락)지연
T0224	BIT/WORD	W10 RH 차종감지 이상 지연
T0314	BIT/WORD	W20-3 LH 로보트 간섭무지연
T0413	BIT/WORD	W20-2 RH 로보트 간섭무지연
T0414	BIT/WORD	W20-3 RH 로보트 간섭무지연
T0516	BIT/WORD	W30 파트이상 (누락)지연
K00100	BIT	W10 LH 파트 로딩완료
P12131	BIT	R21 H/D1 (OT34)
P1211C	BIT	R21 H/D1 (OT13) W20-2 LH 로딩완료
P1211E	BIT	R21 H/D1 (OT15) W20-3 LH 로딩완료
P12115	BIT	R21 H/D1 (OT06)
P12116	BIT	R21 H/D1 (OT07)
P12117	BIT	R21 H/D1 (OT08)
M00071	BIT	OP1 Robot21 Gripper Error
M00072	BIT	OP1 Robot21 Part Error
D150011.2	BIT	OP2 W150 Select Pb
T0724	BIT/WORD	W100 차종감지 이상 지연
P1031A	BIT	R03 (OT11) W100 3차 용접완료
P1041A	BIT	R04 (OT11) W100 3차 용접완료
P1221A	BIT	R22 H/D2 (OT11)
M00841	BIT	W150-1 로딩 로보트 간섭무
T0904	BIT/WORD	W200 작업자 안전확보 이상지연
T0905	BIT/WORD	W200 상.하부 동시감지 시간지연
T0924	BIT/WORD	W200 차종감지 이상 지연
T0994	BIT/WORD	W200 에어블로우 이상
M01084	BIT	W250 4차 기동완료
M01306	BIT	W450 서보 동작가능
M0130B	BIT	W450 상부 안전센서 정상
M0130C	BIT	W450 하부 안전세서 정상
M0130D	BIT	W450 안전매트 정상
M01360	BIT	W450 원위치복귀 Pb (XP)
M01374	BIT	W450 4차 기동
M0137A	BIT	W450 2차 작업준비
M01384	BIT	W450 4차 기동완료
T1303	BIT/WORD	W450 Air Blow On TMR
T1316	BIT/WORD	W450 파트이상 (누락)지연
T1318	BIT/WORD	W450 서보 위치이상 지연
T1319	BIT/WORD	W450 서보 근접센서 위치이상 Tmr
T2211	BIT/WORD	R06 누설가스 검출이상
D12064	WORD	R06 가스 하한
D12068	WORD	R06 가스 상한
D12066	WORD	R06 용접중 가스 유량
M03911	BIT	R06 누설가스 검출이상
P10611	BIT	R06 (OT02)
P10511	BIT	R05 (OT02)
T3101	BIT/WORD	Data Pc Off Error
T3100	BIT/WORD	Data Pc Signal Reset
P1222F	BIT	R22 H/D2 (OT32)
P1232F	BIT	R23 H/D3 (OT32)
P1242F	BIT	R24 H/D4 (OT32)
M05106	BIT	R06 지그 작업중
M05101	BIT	R01 로보트 티치전환
M05102	BIT	R02 로보트 티치전환
T1103	BIT/WORD	W300 Air Blow On TMR
T1116	BIT/WORD	W300 파트이상 (누락)지연
T1118	BIT/WORD	W300 서보 위치이상 지연
T1119	BIT/WORD	W300 서보 근접센서 위치이상 Tmr
K01102	BIT	W300 2차 작업완료
M01106	BIT	W300 서보 동작가능
M01174	BIT	W300 4차 기동
M0117A	BIT	W300 2차 작업준비
M01184	BIT	W300 4차 기동완료
T1203	BIT/WORD	W400 Air Blow On TMR
T1216	BIT/WORD	W400 파트이상 (누락)지연
T1219	BIT/WORD	W400 서보 근접센서 위치이상 Tmr
M01206	BIT	W400 서보 동작가능
M01274	BIT	W400 4차 기동
M0127A	BIT	W400 2차 작업준비
M01284	BIT	W400 4차 기동완료
M0140B	BIT	W130 상부 안전센서 정상
M0140C	BIT	W130 하부 안전세서 정상
M0140D	BIT	W130 안전매트 정상
M01420	BIT	W130 파트없음
M01460	BIT	W130 원위치복귀 Pb (XP)
M01474	BIT	W130 4차 기동
M0147A	BIT	W130 2차 작업준비
M01484	BIT	W130 4차 기동완료
T1403	BIT/WORD	W130 Air Blow On TMR
T1416	BIT/WORD	W130 파트이상 (누락)지연
T1418	BIT/WORD	W130 서보 위치이상 지연
T1419	BIT/WORD	W130 서보 근접센서 위치이상 Tmr
T1420	BIT/WORD	W130 파트없음 지연
T1421	BIT/WORD	W130 파트 OK 지연
P10119	BIT	R01 (OT10)
P1011A	BIT	R01 (OT11)
M0015B	BIT	W10 LH R01 서보 언로딩위치 이동 Pb
P10228	BIT	R02 (OT25)
P10219	BIT	R02 (OT10)
P1021A	BIT	R02 (OT11)
M0025B	BIT	W10 RH R02 서보 언로딩위치 이동 Pb
P10111	BIT	R01 (OT02)
P10112	BIT	R01 (OT03)
P10113	BIT	R01 (OT04)
P10114	BIT	R01 (OT05)
P10115	BIT	R01 (OT06)
P10116	BIT	R01 (OT07)
P10117	BIT	R01 (OT08)
P1011B	BIT	R01 (OT12)
P1011C	BIT	R01 (OT13)
P1011D	BIT	R01 (OT14)
P1011E	BIT	R01 (OT15)
P1011F	BIT	R01 (OT16)
P10120	BIT	R01 (OT17)
P10121	BIT	R01 (OT18)
P10122	BIT	R01 (OT19)
P10123	BIT	R01 (OT20)
P10124	BIT	R01 (OT21)
P10125	BIT	R01 (OT22)
P10126	BIT	R01 (OT23)
P10127	BIT	R01 (OT24)
P1012A	BIT	R01 (OT27)
P1012B	BIT	R01 (OT28)
P1012C	BIT	R01 (OT29)
P1012D	BIT	R01 (OT30)
P1012E	BIT	R01 (OT31)
P10132	BIT	R01 (OT35)
P10133	BIT	R01 (OT36)
P10134	BIT	R01 (OT37)
P10135	BIT	R01 (OT38)
P1013A	BIT	R01 (OT43)
P1013C	BIT	R01 (OT45)
P1013E	BIT	R01 (OT47)
P1013F	BIT	R01 (OT48)
P10140	BIT	R01 (OT49)
P10141	BIT	R01 (OT50)
P10142	BIT	R01 (OT51)
P10143	BIT	R01 (OT52)
P10144	BIT	R01 (OT53)
P10145	BIT	R01 (OT54)
P10146	BIT	R01 (OT55)
P10147	BIT	R01 (OT56)
P10148	BIT	R01 (OT57)
P10149	BIT	R01 (OT58)
P1014A	BIT	R01 (OT59)
P1014B	BIT	R01 (OT60)
P1014C	BIT	R01 (OT61)
P1014D	BIT	R01 (OT62)
P1014E	BIT	R01 (OT63)
P1014F	BIT	R01 (OT64)
P10211	BIT	R02 (OT02)
P10212	BIT	R02 (OT03)
P10213	BIT	R02 (OT04)
P10214	BIT	R02 (OT05)
P10215	BIT	R02 (OT06)
P10216	BIT	R02 (OT07)
P10217	BIT	R02 (OT08)
P1021B	BIT	R02 (OT12)
P1021C	BIT	R02 (OT13)
P1021D	BIT	R02 (OT14)
P1021E	BIT	R02 (OT15)
P1021F	BIT	R02 (OT16)
P10220	BIT	R02 (OT17)
P10221	BIT	R02 (OT18)
P10222	BIT	R02 (OT19)
P10223	BIT	R02 (OT20)
P10224	BIT	R02 (OT21)
P10225	BIT	R02 (OT22)
P10226	BIT	R02 (OT23)
P10227	BIT	R02 (OT24)
P1022A	BIT	R02 (OT27)
P1022B	BIT	R02 (OT28)
P1022C	BIT	R02 (OT29)
P1022D	BIT	R02 (OT30)
P1022E	BIT	R02 (OT31)
P10232	BIT	R02 (OT35)
P10233	BIT	R02 (OT36)
P10234	BIT	R02 (OT37)
P10235	BIT	R02 (OT38)
P1023A	BIT	R02 (OT43)
P1023C	BIT	R02 (OT45)
P1023E	BIT	R02 (OT47)
P10241	BIT	R02 (OT50)
P10242	BIT	R02 (OT51)
P10243	BIT	R02 (OT52)
P10244	BIT	R02 (OT53)
P10245	BIT	R02 (OT54)
P10246	BIT	R02 (OT55)
P10247	BIT	R02 (OT56)
P10249	BIT	R02 (OT58)
P1024A	BIT	R02 (OT59)
P1024B	BIT	R02 (OT60)
P1024C	BIT	R02 (OT61)
P1024D	BIT	R02 (OT62)
P1024E	BIT	R02 (OT63)
P1024F	BIT	R02 (OT64)
P1020E	BIT	R02 비상정지
P1022F	BIT	R02 (OT32)
P1010E	BIT	R01 비상정지
P10312	BIT	R03 (OT03)
P10313	BIT	R03 (OT04)
P10314	BIT	R03 (OT05)
P10315	BIT	R03 (OT06)
P10316	BIT	R03 (OT07)
P10317	BIT	R03 (OT08)
P1031B	BIT	R03 (OT12)
P1031E	BIT	R03 (OT15)
P1031F	BIT	R03 (OT16)
P10320	BIT	R03 (OT17)
P10321	BIT	R03 (OT18)
P10322	BIT	R03 (OT19)
P10323	BIT	R03 (OT20)
P10324	BIT	R03 (OT21)
P10325	BIT	R03 (OT22)
P10326	BIT	R03 (OT23)
P10327	BIT	R03 (OT24)
P1032C	BIT	R03 (OT29)
P1032E	BIT	R03 (OT31)
P10331	BIT	R03 (OT34)
P10332	BIT	R03 (OT35)
P10333	BIT	R03 (OT36)
P10334	BIT	R03 (OT37)
P10335	BIT	R03 (OT38)
P1033A	BIT	R03 (OT43)
P1033C	BIT	R03 (OT45)
P1033E	BIT	R03 (OT47)
P10341	BIT	R03 (OT50)
P10342	BIT	R03 (OT51)
P10343	BIT	R03 (OT52)
P10344	BIT	R03 (OT53)
P10345	BIT	R03 (OT54)
P10346	BIT	R03 (OT55)
P10347	BIT	R03 (OT56)
P10349	BIT	R03 (OT58)
P1034A	BIT	R03 (OT59)
P1034B	BIT	R03 (OT60)
P1034C	BIT	R03 (OT61)
P1034D	BIT	R03 (OT62)
P1034E	BIT	R03 (OT63)
P1034F	BIT	R03 (OT64)
P10412	BIT	R04 (OT03)
P10413	BIT	R04 (OT04)
P10414	BIT	R04 (OT05)
P10415	BIT	R04 (OT06)
P10416	BIT	R04 (OT07)
P10417	BIT	R04 (OT08)
P1041E	BIT	R04 (OT15)
P1041F	BIT	R04 (OT16)
P10420	BIT	R04 (OT17)
P10421	BIT	R04 (OT18)
P10422	BIT	R04 (OT19)
P10423	BIT	R04 (OT20)
P10424	BIT	R04 (OT21)
P10425	BIT	R04 (OT22)
P10426	BIT	R04 (OT23)
P10427	BIT	R04 (OT24)
P1042E	BIT	R04 (OT31)
P10430	BIT	R04 (OT33)
P10431	BIT	R04 (OT34)
P10432	BIT	R04 (OT35)
P10433	BIT	R04 (OT36)
P10434	BIT	R04 (OT37)
P10435	BIT	R04 (OT38)
P1043A	BIT	R04 (OT43)
P1043C	BIT	R04 (OT45)
P1043E	BIT	R04 (OT47)
P10441	BIT	R04 (OT50)
P10442	BIT	R04 (OT51)
P10443	BIT	R04 (OT52)
P10444	BIT	R04 (OT53)
P10445	BIT	R04 (OT54)
P10446	BIT	R04 (OT55)
P10447	BIT	R04 (OT56)
P10449	BIT	R04 (OT58)
P1044A	BIT	R04 (OT59)
P1044B	BIT	R04 (OT60)
P1044C	BIT	R04 (OT61)
P1044D	BIT	R04 (OT62)
P1044E	BIT	R04 (OT63)
P1044F	BIT	R04 (OT64)
P10512	BIT	R05 (OT03)
P10513	BIT	R05 (OT04)
P10514	BIT	R05 (OT05)
P10515	BIT	R05 (OT06)
P10516	BIT	R05 (OT07)
P10517	BIT	R05 (OT08)
P1051C	BIT	R05 (OT13)
P1051D	BIT	R05 (OT14)
P1051E	BIT	R05 (OT15)
P1051F	BIT	R05 (OT16)
P10520	BIT	R05 (OT17)
P10521	BIT	R05 (OT18)
P10522	BIT	R05 (OT19)
P10523	BIT	R05 (OT20)
P10524	BIT	R05 (OT21)
P10525	BIT	R05 (OT22)
P10526	BIT	R05 (OT23)
P10527	BIT	R05 (OT24)
P1052E	BIT	R05 (OT31)
P10530	BIT	R05 (OT33)
P10531	BIT	R05 (OT34)
P10532	BIT	R05 (OT35)
P10533	BIT	R05 (OT36)
P10534	BIT	R05 (OT37)
P10535	BIT	R05 (OT38)
P1053A	BIT	R05 (OT43)
P1053C	BIT	R05 (OT45)
P1053E	BIT	R05 (OT47)
P10541	BIT	R05 (OT50)
P10542	BIT	R05 (OT51)
P10543	BIT	R05 (OT52)
P10544	BIT	R05 (OT53)
P10545	BIT	R05 (OT54)
P10546	BIT	R05 (OT55)
P10547	BIT	R05 (OT56)
P10549	BIT	R05 (OT58)
P1054A	BIT	R05 (OT59)
P1054B	BIT	R05 (OT60)
P1054C	BIT	R05 (OT61)
P1054D	BIT	R05 (OT62)
P1054E	BIT	R05 (OT63)
P1054F	BIT	R05 (OT64)
P10612	BIT	R06 (OT03)
P10613	BIT	R06 (OT04)
P10614	BIT	R06 (OT05)
P10615	BIT	R06 (OT06)
P10616	BIT	R06 (OT07)
P10617	BIT	R06 (OT08)
P1061C	BIT	R06 (OT13)
P1061D	BIT	R06 (OT14)
P1061E	BIT	R06 (OT15)
P1061F	BIT	R06 (OT16)
P10620	BIT	R06 (OT17)
P10621	BIT	R06 (OT18)
P10622	BIT	R06 (OT19)
P10623	BIT	R06 (OT20)
P10624	BIT	R06 (OT21)
P10625	BIT	R06 (OT22)
P10627	BIT	R06 (OT24)
P1062C	BIT	R06 (OT29)
P10630	BIT	R06 (OT33)
P10631	BIT	R06 (OT34)
P10632	BIT	R06 (OT35)
P10633	BIT	R06 (OT36)
P10634	BIT	R06 (OT37)
P10635	BIT	R06 (OT38)
P1063A	BIT	R06 (OT43)
P1063C	BIT	R06 (OT45)
P1063E	BIT	R06 (OT47)
M10130	BIT	R01 (IN33)
M10131	BIT	R01 (IN34)
M10132	BIT	R01 (IN35)
M10133	BIT	R01 (IN36)
M10134	BIT	R01 (IN37)
M10135	BIT	R01 (IN38) 가스반출 요구
M10139	BIT	R01 (IN42)
M1013A	BIT	R01 (IN43) 노즐커버 체크요구
M1013B	BIT	R01 (IN44)
M1013E	BIT	R01 (IN47)
M1013F	BIT	R01 (IN48)
M10141	BIT	R01 (IN50)
M10142	BIT	R01 (IN51)
M10143	BIT	R01 (IN52)
M10145	BIT	R01 (IN54)
M10146	BIT	R01 (IN55)
M10147	BIT	R01 (IN56)
M10148	BIT	R01 (IN57)
M10149	BIT	R01 (IN58)
M1014A	BIT	R01 (IN59)
M1014B	BIT	R01 (IN60)
M1014C	BIT	R01 (IN61)
M1014D	BIT	R01 (IN62)
M1014E	BIT	R01 (IN63)
M1014F	BIT	R01 (IN64)
M10230	BIT	R02 (IN33)
M10231	BIT	R02 (IN34)
M10232	BIT	R02 (IN35)
M10233	BIT	R02 (IN36)
M10234	BIT	R02 (IN37)
M10235	BIT	R02 (IN38) 가스반출 요구
M10239	BIT	R02 (IN42)
M1023A	BIT	R02 (IN43) 노즐커버 체크요구
M1023B	BIT	R02 (IN44)
M1023E	BIT	R02 (IN47)
M1023F	BIT	R02 (IN48)
M10241	BIT	R02 (IN50)
M10242	BIT	R02 (IN51)
M10243	BIT	R02 (IN52)
M10244	BIT	R02 (IN53)
M10245	BIT	R02 (IN54)
M10246	BIT	R02 (IN55)
M10247	BIT	R02 (IN56)
M10249	BIT	R02 (IN58)
M1024A	BIT	R02 (IN59)
M1024B	BIT	R02 (IN60)
M1024C	BIT	R02 (IN61)
M1024D	BIT	R02 (IN62)
M1024E	BIT	R02 (IN63)
M1024F	BIT	R02 (IN64)
M10144	BIT	R01 (IN53)
M10330	BIT	R03 (IN33)
M10331	BIT	R03 (IN34)
M10332	BIT	R03 (IN35)
M10333	BIT	R03 (IN36)
M10334	BIT	R03 (IN37)
M10335	BIT	R03 (IN38) 가스반출 요구
M10339	BIT	R03 (IN42)
M1033A	BIT	R03 (IN43) 노즐커버 체크요구
M1033B	BIT	R03 (IN44)
M1033E	BIT	R03 (IN47)
M1033F	BIT	R03 (IN48)
M10341	BIT	R03 (IN50)
M10342	BIT	R03 (IN51)
M10343	BIT	R03 (IN52)
M10344	BIT	R03 (IN53)
M10345	BIT	R03 (IN54)
M10346	BIT	R03 (IN55)
M10347	BIT	R03 (IN56)
M10349	BIT	R03 (IN58)
M1034A	BIT	R03 (IN59)
M1034B	BIT	R03 (IN60)
M1034C	BIT	R03 (IN61)
M1034D	BIT	R03 (IN62)
M1034E	BIT	R03 (IN63)
M1034F	BIT	R03 (IN64)
M10430	BIT	R04 (IN33)
M10431	BIT	R04 (IN34)
M10432	BIT	R04 (IN35)
M10433	BIT	R04 (IN36)
M10434	BIT	R04 (IN37)
M10435	BIT	R04 (IN38) 가스반출 요구
M10439	BIT	R04 (IN42)
M1043A	BIT	R04 (IN43) 노즐커버 체크요구
M1043B	BIT	R04 (IN44)
M1043E	BIT	R04 (IN47)
M1043F	BIT	R04 (IN48)
M10441	BIT	R04 (IN50)
M10442	BIT	R04 (IN51)
M10443	BIT	R04 (IN52)
M10444	BIT	R04 (IN53)
M10445	BIT	R04 (IN54)
M10446	BIT	R04 (IN55)
M10447	BIT	R04 (IN56)
M10449	BIT	R04 (IN58)
M1044A	BIT	R04 (IN59)
M1044B	BIT	R04 (IN60)
M1044C	BIT	R04 (IN61)
M1044D	BIT	R04 (IN62)
M1044E	BIT	R04 (IN63)
M1044F	BIT	R04 (IN64)
M10530	BIT	R05 (IN33)
M10531	BIT	R05 (IN34)
M10532	BIT	R05 (IN35)
M10533	BIT	R05 (IN36)
M10534	BIT	R05 (IN37)
M10535	BIT	R05 (IN38) 가스반출 요구
M10539	BIT	R05 (IN42)
M1053A	BIT	R05 (IN43) 노즐커버 체크요구
M1053B	BIT	R05 (IN44)
M1053E	BIT	R05 (IN47)
M1053F	BIT	R05 (IN48)
M10541	BIT	R05 (IN50)
M10542	BIT	R05 (IN51)
M10543	BIT	R05 (IN52)
M10544	BIT	R05 (IN53)
M10545	BIT	R05 (IN54)
M10546	BIT	R05 (IN55)
M10547	BIT	R05 (IN56)
M10549	BIT	R05 (IN58)
M1054A	BIT	R05 (IN59)
M1054B	BIT	R05 (IN60)
M1054C	BIT	R05 (IN61)
M1054D	BIT	R05 (IN62)
M1054E	BIT	R05 (IN63)
M1054F	BIT	R05 (IN64)
M10630	BIT	R06 (IN33)
M10631	BIT	R06 (IN34)
M10632	BIT	R06 (IN35)
M10633	BIT	R06 (IN36)
M10634	BIT	R06 (IN37)
M10635	BIT	R06 (IN38) 가스반출 요구
M10639	BIT	R06 (IN42)
M1063A	BIT	R06 (IN43) 노즐커버 체크요구
M1063B	BIT	R06 (IN44)
M1063E	BIT	R06 (IN47)
M1063F	BIT	R06 (IN48)
P1222C	BIT	R22 H/D2 (OT29)
M1214A	BIT	R21 H/D1 (IN59)
M1214B	BIT	R21 H/D1 (IN60)
M1214C	BIT	R21 H/D1 (IN61)
M1214D	BIT	R21 H/D1 (IN62)
M1214E	BIT	R21 H/D1 (IN63)
M1214F	BIT	R21 H/D1 (IN64)
M12152	BIT	R21 H/D1 (IN67)
M12153	BIT	R21 H/D1 (IN68)
M12154	BIT	R21 H/D1 (IN69)
M12155	BIT	R21 H/D1 (IN70)
M12156	BIT	R21 H/D1 (IN71)
M12157	BIT	R21 H/D1 (IN72)
M12158	BIT	R21 H/D1 (IN73)
M12159	BIT	R21 H/D1 (IN74)
M1215A	BIT	R21 H/D1 (IN75)
M1215B	BIT	R21 H/D1 (IN76)
M1215C	BIT	R21 H/D1 (IN77)
M1215D	BIT	R21 H/D1 (IN78)
M1215E	BIT	R21 H/D1 (IN79)
M1215F	BIT	R21 H/D1 (IN80)
M12160	BIT	R21 H/D1 (IN81)
M12161	BIT	R21 H/D1 (IN82)
M12162	BIT	R21 H/D1 (IN83)
M12163	BIT	R21 H/D1 (IN84)
M12164	BIT	R21 H/D1 (IN85)
M12165	BIT	R21 H/D1 (IN86)
M12166	BIT	R21 H/D1 (IN87)
M12167	BIT	R21 H/D1 (IN88)
M12168	BIT	R21 H/D1 (IN89)
M12169	BIT	R21 H/D1 (IN90)
M1216A	BIT	R21 H/D1 (IN91)
M1216B	BIT	R21 H/D1 (IN92)
M1216C	BIT	R21 H/D1 (IN93)
M1216D	BIT	R21 H/D1 (IN94)
M1216E	BIT	R21 H/D1 (IN95)
M1216F	BIT	R21 H/D1 (IN96)
P12127	BIT	R21 H/D1 (OT24)
P1212A	BIT	R21 H/D1 (OT27)
P1212C	BIT	R21 H/D1 (OT29)
P1212D	BIT	R21 H/D1 (OT30)
P1212E	BIT	R21 H/D1 (OT31)
P1212F	BIT	R21 H/D1 (OT32)
P1213A	BIT	R21 H/D1 (OT43)
P1213B	BIT	R21 H/D1 (OT44)
P1213C	BIT	R21 H/D1 (OT45)
P1213D	BIT	R21 H/D1 (OT46)
P1213E	BIT	R21 H/D1 (OT47)
P1213F	BIT	R21 H/D1 (OT48)
P1214A	BIT	R21 H/D1 (OT59)
P1214B	BIT	R21 H/D1 (OT60)
P1214C	BIT	R21 H/D1 (OT61)
P1214D	BIT	R21 H/D1 (OT62)
P1214E	BIT	R21 H/D1 (OT63)
P1214F	BIT	R21 H/D1 (OT64)
P12150	BIT	R21 H/D1 (OT65)
P12151	BIT	R21 H/D1 (OT66)
P12152	BIT	R21 H/D1 (OT67)
P12153	BIT	R21 H/D1 (OT68)
P12154	BIT	R21 H/D1 (OT69)
P12155	BIT	R21 H/D1 (OT70)
P12156	BIT	R21 H/D1 (OT71)
P12157	BIT	R21 H/D1 (OT72)
P12158	BIT	R21 H/D1 (OT73)
P12159	BIT	R21 H/D1 (OT74)
P1215A	BIT	R21 H/D1 (OT75)
P1215B	BIT	R21 H/D1 (OT76)
P1215C	BIT	R21 H/D1 (OT77)
P1215D	BIT	R21 H/D1 (OT78)
P1215E	BIT	R21 H/D1 (OT79)
P1215F	BIT	R21 H/D1 (OT80)
P12160	BIT	R21 H/D1 (OT81)
P12161	BIT	R21 H/D1 (OT82)
P12162	BIT	R21 H/D1 (OT83)
P12163	BIT	R21 H/D1 (OT84)
P12164	BIT	R21 H/D1 (OT85)
P12165	BIT	R21 H/D1 (OT86)
P12166	BIT	R21 H/D1 (OT87)
P12167	BIT	R21 H/D1 (OT88)
P12168	BIT	R21 H/D1 (OT89)
P12169	BIT	R21 H/D1 (OT90)
P1216A	BIT	R21 H/D1 (OT91)
P1216B	BIT	R21 H/D1 (OT92)
P1216C	BIT	R21 H/D1 (OT93)
P1216D	BIT	R21 H/D1 (OT94)
P1216E	BIT	R21 H/D1 (OT95)
P1216F	BIT	R21 H/D1 (OT96)
P12212	BIT	R22 H/D2 (OT03)
P12213	BIT	R22 H/D2 (OT04)
P12214	BIT	R22 H/D2 (OT05)
P12215	BIT	R22 H/D2 (OT06)
P12216	BIT	R22 H/D2 (OT07)
P12217	BIT	R22 H/D2 (OT08)
P1221B	BIT	R22 H/D2 (OT12)
P1221C	BIT	R22 H/D2 (OT13)
P1221D	BIT	R22 H/D2 (OT14)
P1221E	BIT	R22 H/D2 (OT15)
P1221F	BIT	R22 H/D2 (OT16)
P12220	BIT	R22 H/D2 (OT17)
P12221	BIT	R22 H/D2 (OT18)
P12222	BIT	R22 H/D2 (OT19)
P12223	BIT	R22 H/D2 (OT20)
P12224	BIT	R22 H/D2 (OT21)
P12225	BIT	R22 H/D2 (OT22)
P12226	BIT	R22 H/D2 (OT23)
P12227	BIT	R22 H/D2 (OT24)
P1222D	BIT	R22 H/D2 (OT30)
P1222E	BIT	R22 H/D2 (OT31)
P12230	BIT	R22 H/D2 (OT33)
P12231	BIT	R22 H/D2 (OT34)
P12232	BIT	R22 H/D2 (OT35)
P12233	BIT	R22 H/D2 (OT36)
P12234	BIT	R22 H/D2 (OT37)
P12235	BIT	R22 H/D2 (OT38)
P12236	BIT	R22 H/D2 (OT39)
P12237	BIT	R22 H/D2 (OT40)
P12238	BIT	R22 H/D2 (OT41)
P12239	BIT	R22 H/D2 (OT42)
P1223A	BIT	R22 H/D2 (OT43)
P1223B	BIT	R22 H/D2 (OT44)
P1223C	BIT	R22 H/D2 (OT45)
P1223D	BIT	R22 H/D2 (OT46)
P1223E	BIT	R22 H/D2 (OT47)
P1223F	BIT	R22 H/D2 (OT48)
P1224A	BIT	R22 H/D2 (OT59)
P1224B	BIT	R22 H/D2 (OT60)
P1224C	BIT	R22 H/D2 (OT61)
P1224D	BIT	R22 H/D2 (OT62)
P1224E	BIT	R22 H/D2 (OT63)
P1224F	BIT	R22 H/D2 (OT64)
P12250	BIT	R22 H/D2 (OT65)
P12251	BIT	R22 H/D2 (OT66)
P12252	BIT	R22 H/D2 (OT67)
P12253	BIT	R22 H/D2 (OT68)
P12254	BIT	R22 H/D2 (OT69)
P12255	BIT	R22 H/D2 (OT70)
P12256	BIT	R22 H/D2 (OT71)
P12257	BIT	R22 H/D2 (OT72)
P12258	BIT	R22 H/D2 (OT73)
P12259	BIT	R22 H/D2 (OT74)
P1225A	BIT	R22 H/D2 (OT75)
P1225B	BIT	R22 H/D2 (OT76)
P1225C	BIT	R22 H/D2 (OT77)
P1225D	BIT	R22 H/D2 (OT78)
P1225E	BIT	R22 H/D2 (OT79)
P1225F	BIT	R22 H/D2 (OT80)
P12260	BIT	R22 H/D2 (OT81)
P12261	BIT	R22 H/D2 (OT82)
P12262	BIT	R22 H/D2 (OT83)
P12263	BIT	R22 H/D2 (OT84)
P12264	BIT	R22 H/D2 (OT85)
P12265	BIT	R22 H/D2 (OT86)
P12266	BIT	R22 H/D2 (OT87)
P12267	BIT	R22 H/D2 (OT88)
P12268	BIT	R22 H/D2 (OT89)
P12269	BIT	R22 H/D2 (OT90)
P1226A	BIT	R22 H/D2 (OT91)
P1226B	BIT	R22 H/D2 (OT92)
P1226C	BIT	R22 H/D2 (OT93)
P1226D	BIT	R22 H/D2 (OT94)
P1226E	BIT	R22 H/D2 (OT95)
P1226F	BIT	R22 H/D2 (OT96)
M1224A	BIT	R22 H/D2 (IN59)
M1224B	BIT	R22 H/D2 (IN60)
M1224C	BIT	R22 H/D2 (IN61)
M1224D	BIT	R22 H/D2 (IN62)
M1224E	BIT	R22 H/D2 (IN63)
M1224F	BIT	R22 H/D2 (IN64)
M12250	BIT	R22 H/D2 (IN65)
M12251	BIT	R22 H/D2 (IN66)
M12252	BIT	R22 H/D2 (IN67)
M12253	BIT	R22 H/D2 (IN68)
M12254	BIT	R22 H/D2 (IN69)
M12255	BIT	R22 H/D2 (IN70)
M12256	BIT	R22 H/D2 (IN71)
M12257	BIT	R22 H/D2 (IN72)
M12258	BIT	R22 H/D2 (IN73)
M12259	BIT	R22 H/D2 (IN74)
M1225A	BIT	R22 H/D2 (IN75)
M1225B	BIT	R22 H/D2 (IN76)
M1225C	BIT	R22 H/D2 (IN77)
M1225D	BIT	R22 H/D2 (IN78)
M1225E	BIT	R22 H/D2 (IN79)
M1225F	BIT	R22 H/D2 (IN80)
M12260	BIT	R22 H/D2 (IN81)
M12261	BIT	R22 H/D2 (IN82)
M12262	BIT	R22 H/D2 (IN83)
M12263	BIT	R22 H/D2 (IN84)
M12264	BIT	R22 H/D2 (IN85)
M12265	BIT	R22 H/D2 (IN86)
M12266	BIT	R22 H/D2 (IN87)
M12267	BIT	R22 H/D2 (IN88)
M12268	BIT	R22 H/D2 (IN89)
M12269	BIT	R22 H/D2 (IN90)
M1226A	BIT	R22 H/D2 (IN91)
M1226B	BIT	R22 H/D2 (IN92)
M1226C	BIT	R22 H/D2 (IN93)
M1226D	BIT	R22 H/D2 (IN94)
M1226E	BIT	R22 H/D2 (IN95)
M1226F	BIT	R22 H/D2 (IN96)
P12317	BIT	R23 H/D3 (OT08)
P12319	BIT	R23 H/D3 (OT10)
P1231A	BIT	R23 H/D3 (OT11)
P1232A	BIT	R23 H/D3 (OT27)
P12332	BIT	R23 H/D3 (OT35)
P12333	BIT	R23 H/D3 (OT36)
P12334	BIT	R23 H/D3 (OT37)
P12335	BIT	R23 H/D3 (OT38)
P12336	BIT	R23 H/D3 (OT39)
P12337	BIT	R23 H/D3 (OT40)
P12338	BIT	R23 H/D3 (OT41)
P12339	BIT	R23 H/D3 (OT42)
P1233A	BIT	R23 H/D3 (OT43)
P1233B	BIT	R23 H/D3 (OT44)
P1233C	BIT	R23 H/D3 (OT45)
P1233D	BIT	R23 H/D3 (OT46)
P1233E	BIT	R23 H/D3 (OT47)
P1233F	BIT	R23 H/D3 (OT48)
P1234A	BIT	R23 H/D3 (OT59)
P1234B	BIT	R23 H/D3 (OT60)
P1234C	BIT	R23 H/D3 (OT61)
P1234D	BIT	R23 H/D3 (OT62)
P1234E	BIT	R23 H/D3 (OT63)
P1234F	BIT	R23 H/D3 (OT64)
P12350	BIT	R23 H/D3 (OT65)
P12351	BIT	R23 H/D3 (OT66)
P12352	BIT	R23 H/D3 (OT67)
P12353	BIT	R23 H/D3 (OT68)
P12354	BIT	R23 H/D3 (OT69)
P12355	BIT	R23 H/D3 (OT70)
P12356	BIT	R23 H/D3 (OT71)
P12357	BIT	R23 H/D3 (OT72)
P12358	BIT	R23 H/D3 (OT73)
P12359	BIT	R23 H/D3 (OT74)
P1235A	BIT	R23 H/D3 (OT75)
P1235B	BIT	R23 H/D3 (OT76)
P1235C	BIT	R23 H/D3 (OT77)
P1235D	BIT	R23 H/D3 (OT78)
P1235E	BIT	R23 H/D3 (OT79)
P1235F	BIT	R23 H/D3 (OT80)
P12360	BIT	R23 H/D3 (OT81)
P12361	BIT	R23 H/D3 (OT82)
P12362	BIT	R23 H/D3 (OT83)
P12363	BIT	R23 H/D3 (OT84)
P12364	BIT	R23 H/D3 (OT85)
P12365	BIT	R23 H/D3 (OT86)
P12366	BIT	R23 H/D3 (OT87)
P12367	BIT	R23 H/D3 (OT88)
P12368	BIT	R23 H/D3 (OT89)
P12369	BIT	R23 H/D3 (OT90)
P1236A	BIT	R23 H/D3 (OT91)
P1236B	BIT	R23 H/D3 (OT92)
P1236C	BIT	R23 H/D3 (OT93)
P1236D	BIT	R23 H/D3 (OT94)
P1236E	BIT	R23 H/D3 (OT95)
P1236F	BIT	R23 H/D3 (OT96)
M1234A	BIT	R23 H/D3 (IN59)
M1234B	BIT	R23 H/D3 (IN60)
M1234C	BIT	R23 H/D3 (IN61)
M1234D	BIT	R23 H/D3 (IN62)
M1234E	BIT	R23 H/D3 (IN63)
M1234F	BIT	R23 H/D3 (IN64)
M12350	BIT	R23 H/D3 (IN65)
M12351	BIT	R23 H/D3 (IN66)
M12352	BIT	R23 H/D3 (IN67)
M12353	BIT	R23 H/D3 (IN68)
M12354	BIT	R23 H/D3 (IN69)
M12355	BIT	R23 H/D3 (IN70)
M12356	BIT	R23 H/D3 (IN71)
M12357	BIT	R23 H/D3 (IN72)
M12358	BIT	R23 H/D3 (IN73)
M12359	BIT	R23 H/D3 (IN74)
M1235A	BIT	R23 H/D3 (IN75)
M1235B	BIT	R23 H/D3 (IN76)
M1235C	BIT	R23 H/D3 (IN77)
M1235D	BIT	R23 H/D3 (IN78)
M1235E	BIT	R23 H/D3 (IN79)
M1235F	BIT	R23 H/D3 (IN80)
M12360	BIT	R23 H/D3 (IN81)
M12361	BIT	R23 H/D3 (IN82)
M12362	BIT	R23 H/D3 (IN83)
M12363	BIT	R23 H/D3 (IN84)
M12364	BIT	R23 H/D3 (IN85)
M12365	BIT	R23 H/D3 (IN86)
M12366	BIT	R23 H/D3 (IN87)
M12367	BIT	R23 H/D3 (IN88)
M12368	BIT	R23 H/D3 (IN89)
M12369	BIT	R23 H/D3 (IN90)
M1236A	BIT	R23 H/D3 (IN91)
M1236B	BIT	R23 H/D3 (IN92)
M1236C	BIT	R23 H/D3 (IN93)
M1236D	BIT	R23 H/D3 (IN94)
M1236E	BIT	R23 H/D3 (IN95)
M1236F	BIT	R23 H/D3 (IN96)
M1244A	BIT	R24 H/D4 (IN59)
M1244B	BIT	R24 H/D4 (IN60)
M1244C	BIT	R24 H/D4 (IN61)
M1244D	BIT	R24 H/D4 (IN62)
M1244E	BIT	R24 H/D4 (IN63)
M1244F	BIT	R24 H/D4 (IN64)
M12454	BIT	R24 H/D4 (IN69)
M12455	BIT	R24 H/D4 (IN70)
M12456	BIT	R24 H/D4 (IN71)
M12457	BIT	R24 H/D4 (IN72)
M1245C	BIT	R24 H/D4 (IN77)
M1245D	BIT	R24 H/D4 (IN78)
M1245E	BIT	R24 H/D4 (IN79)
M1245F	BIT	R24 H/D4 (IN80)
M12464	BIT	R24 H/D4 (IN85)
M12465	BIT	R24 H/D4 (IN86)
M12466	BIT	R24 H/D4 (IN87)
M12467	BIT	R24 H/D4 (IN88)
M12468	BIT	R24 H/D4 (IN89)
M12469	BIT	R24 H/D4 (IN90)
M1246A	BIT	R24 H/D4 (IN91)
M1246B	BIT	R24 H/D4 (IN92)
M1246C	BIT	R24 H/D4 (IN93)
M1246D	BIT	R24 H/D4 (IN94)
M1246E	BIT	R24 H/D4 (IN95)
M1246F	BIT	R24 H/D4 (IN96)
P12417	BIT	R24 H/D4 (OT08)
P1241F	BIT	R24 H/D4 (OT16)
P12428	BIT	R24 H/D4 (OT25)
P1242A	BIT	R24 H/D4 (OT27)
P1242B	BIT	R24 H/D4 (OT28)
P1242C	BIT	R24 H/D4 (OT29)
P1242D	BIT	R24 H/D4 (OT30)
P1242E	BIT	R24 H/D4 (OT31)
P12430	BIT	R24 H/D4 (OT33) 마스타 언로딩완료
P12433	BIT	R24 H/D4 (OT36)
P12434	BIT	R24 H/D4 (OT37)
P12438	BIT	R24 H/D4 (OT41)
P12439	BIT	R24 H/D4 (OT42)
P1243A	BIT	R24 H/D4 (OT43)
P1243B	BIT	R24 H/D4 (OT44)
P1243C	BIT	R24 H/D4 (OT45)
P1243D	BIT	R24 H/D4 (OT46)
P1243E	BIT	R24 H/D4 (OT47)
P1243F	BIT	R24 H/D4 (OT48)
P12445	BIT	R24 H/D4 (OT54)
P12446	BIT	R24 H/D4 (OT55)
P12447	BIT	R24 H/D4 (OT56)
P12448	BIT	R24 H/D4 (OT57)
P12449	BIT	R24 H/D4 (OT58)
P1244A	BIT	R24 H/D4 (OT59)
P1244B	BIT	R24 H/D4 (OT60)
P1244C	BIT	R24 H/D4 (OT61)
P1244D	BIT	R24 H/D4 (OT62)
P1244E	BIT	R24 H/D4 (OT63)
P1244F	BIT	R24 H/D4 (OT64)
P12450	BIT	R24 H/D4 (OT65)
P12451	BIT	R24 H/D4 (OT66)
P12452	BIT	R24 H/D4 (OT67)
P12453	BIT	R24 H/D4 (OT68)
P12454	BIT	R24 H/D4 (OT69)
P12455	BIT	R24 H/D4 (OT70)
P12456	BIT	R24 H/D4 (OT71)
P12457	BIT	R24 H/D4 (OT72)
P12458	BIT	R24 H/D4 (OT73)
P12459	BIT	R24 H/D4 (OT74)
P1245A	BIT	R24 H/D4 (OT75)
P1245B	BIT	R24 H/D4 (OT76)
P1245C	BIT	R24 H/D4 (OT77)
P1245D	BIT	R24 H/D4 (OT78)
P1245E	BIT	R24 H/D4 (OT79)
P1245F	BIT	R24 H/D4 (OT80)
P12460	BIT	R24 H/D4 (OT81)
P12461	BIT	R24 H/D4 (OT82)
P12462	BIT	R24 H/D4 (OT83)
P12463	BIT	R24 H/D4 (OT84)
P12464	BIT	R24 H/D4 (OT85)
P12465	BIT	R24 H/D4 (OT86)
P12466	BIT	R24 H/D4 (OT87)
P12467	BIT	R24 H/D4 (OT88)
P12468	BIT	R24 H/D4 (OT89)
P12469	BIT	R24 H/D4 (OT90)
P1246A	BIT	R24 H/D4 (OT91)
P1246B	BIT	R24 H/D4 (OT92)
P1246C	BIT	R24 H/D4 (OT93)
P1246D	BIT	R24 H/D4 (OT94)
P1246E	BIT	R24 H/D4 (OT95)
P1246F	BIT	R24 H/D4 (OT96)
M0001F	BIT	임시 접점
M00074	BIT	OP2 Robot22 Gripper Error
M00075	BIT	OP2 Robot23 Gripper Error
K00116	BIT	W10 LH 핀하강 요구
P12130	BIT	R21 H/D1 (OT33)
D15014.9	BIT	W300 측정 [동도] 판정 선택 데이터 ON=PLC판정 OFF=동도판정
D15002.3	BIT	W300 동도체크 바이페스
K01142	BIT	G2: FRT LH "T" 측정 OK
K01143	BIT	G3: FRT LH "L" 측정 OK
K01144	BIT	G4: FRT LH "H" 측정 OK
K01145	BIT	G5: FRT RH "T" 측정 OK
K01146	BIT	G6: FRT RH "L" 측정 OK
K01147	BIT	G7: FRT RH "H" 측정 OK
K01148	BIT	G8: RR LH "T" 측정 OK
K01149	BIT	G9: RR LH "L" 측정 OK
K0114A	BIT	G10: RR LH "H" 측정 OK
K0114B	BIT	G11: RR RH "T" 측정 OK
K0114C	BIT	G12: RR RH "L" 측정 OK
K0114D	BIT	G13: RR RH "H" 측정 OK
K01152	BIT	G2: FRT LH "T" 측정 NG
K01153	BIT	G3: FRT LH "L" 측정 NG
K01154	BIT	G4: FRT LH "H" 측정 NG
K01155	BIT	G5: FRT RH "T" 측정 NG
K01156	BIT	G6: FRT RH "L" 측정 NG
K01157	BIT	G7: FRT RH "H" 측정 NG
K01158	BIT	G8: RR LH "T" 측정 NG
K01159	BIT	G9: RR LH "L" 측정 NG
K0115A	BIT	G10: RR LH "H" 측정 NG
K0115B	BIT	G11: RR RH "T" 측정 NG
K0115C	BIT	G12: RR RH "L" 측정 NG
K0115D	BIT	G13: RR RH "H" 측정 NG
D01171	WORD	W300 G1 측정 1:OK 2:NG
D01172	WORD	W300 G2 측정 1:OK 2:NG
D01173	WORD	W300 G3 측정 1:OK 2:NG
D01174	WORD	W300 G4 측정 1:OK 2:NG
D01175	WORD	W300 G5 측정 1:OK 2:NG
D01176	WORD	W300 G6 측정 1:OK 2:NG
D01177	WORD	W300 G7 측정 1:OK 2:NG
D01178	WORD	W300 G8 측정 1:OK 2:NG
D01179	WORD	W300 G9 측정 1:OK 2:NG
D01180	WORD	W300 G10 측정 1:OK 2:NG
D01181	WORD	W300 G11 측정 1:OK 2:NG
D01182	WORD	W300 G12 측정 1:OK 2:NG
D01183	WORD	W300 G13 측정 1:OK 2:NG
T4126	BIT/WORD	W400 작업자 NG 취출기동 
D00717	WORD	W100 파트램프 상태7
P00337	BIT	W10 LH 2차 클램프 잠김
P00336	BIT	W10 LH 2차 클램프 풀림
P00537	BIT	W10 RH 2차 클램프 잠김
P00536	BIT	W10 RH 2차 클램프 풀림
T1493	BIT/WORD	W130 스캐너 TRIGGER 차단
K0140A	BIT	W130 Scan Data OK
K0140B	BIT	W130 Scan Data NG
T1492	BIT/WORD	W130 스캐너 트리거 완료 지연
M0149E	BIT	W130 스캐너 트리거 완료
K01431	BIT	W130 2차 스캔 OK
K01432	BIT	W130 2차 스캔 NG
M0150B	BIT	W480 상부 안전센서 정상
M0150C	BIT	W480 하부 안전세서 정상
M0150D	BIT	W480 안전매트 정상
M01560	BIT	W480 원위치복귀 Pb (XP)
M01574	BIT	W480 4차 기동
M0157A	BIT	W480 2차 작업준비
M01584	BIT	W480 4차 기동완료
M0159E	BIT	W480 스캐너 트리거 완료
T1503	BIT/WORD	W480 Air Blow On TMR
T1516	BIT/WORD	W480 파트이상 (누락)지연
T1518	BIT/WORD	W480 서보 위치이상 지연
T1519	BIT/WORD	W480 서보 근접센서 위치이상 Tmr
T1520	BIT/WORD	W480 파트없음 지연
T1521	BIT/WORD	W480 파트 OK 지연
T1592	BIT/WORD	W480 스캐너 트리거 완료 지연
T1593	BIT/WORD	W480 스캐너 TRIGGER 차단
K0150A	BIT	W480 Scan Data OK
K0150B	BIT	W480 Scan Data NG
K01531	BIT	W480 2차 스캔 OK
K01532	BIT	W480 2차 스캔 NG
T1408	BIT/WORD	W130 1차 스캔 NG지연
T1409	BIT/WORD	W130 2차 스캔 NG지연
D11000	WORD	W130 1차 스캔 DATA AUX
D11100	WORD	W130 2차 스캔 DATA AUX
D13150.0	BIT	R01 용접 누락확인 OK
D13151.0	BIT	R02 용접 누락확인 OK
D13152.0	BIT	R03 용접 누락확인 OK
D13153.0	BIT	R04 용접 누락확인 OK
D13154.0	BIT	R05 용접 누락확인 OK
D13155.0	BIT	R06 용접 누락확인 OK
M0109F	BIT	W400 제품 NG 데이터
M04992	BIT	절전
M04240	BIT	NG-PLT 래치확인 진입보조
P01718	BIT	NG-PLT 래치감지 1-1
P01719	BIT	NG-PLT 래치감지 1-2
P0171A	BIT	NG-PLT 래치감지 2-1
P0171B	BIT	NG-PLT 래치감지 2-2
P0171C	BIT	NG-PLT 래치감지 3-1
P0171D	BIT	NG-PLT 래치감지 3-2
P0171E	BIT	NG-PLT 래치감지 4-1
P0171F	BIT	NG-PLT 래치감지 4-2
T4204	BIT/WORD	NG-PLT 푸셔 전진
P01720	BIT	NG-PLT 푸샤 전진 [SOL]
P01721	BIT	NG-PLT 푸샤 후진 [SOL]
P0170A	BIT	NG-PLT 푸샤 전진기동
T4205	BIT/WORD	NG-PLT 푸셔 후진
P01700	BIT	NG-PLT 푸샤 전진단
P01701	BIT	NG-PLT 푸샤 후진단
T4240	BIT/WORD	NG-PLT 래치1 확인
T4241	BIT/WORD	NG-PLT 래치2 확인
T4242	BIT/WORD	NG-PLT 래치3 확인
D18554	WORD	W450 -> H/D4 차종버퍼
D27020	WORD	W130 스케너 data Aux_RH
D27520	WORD	W480 스케너 data Aux_RH
R11000	WORD	W10 LH R01 용접시간 저장 시작워드
R11099	WORD	W10 LH R01 용접시간 저장 시작워드
K00001	BIT	차종.1 JG
D13102.2	BIT	PLC -> PC Car Type-2
D13102.3	BIT	PLC -> PC Car Type-3
D13102.4	BIT	PLC -> PC Car Type-4
D118000	WORD	W480 -> R24 DATA 전송
D111052	WORD	PLC -> PC 동도 DATA 판정
D154603	WORD	W300 동도 버퍼
M0499A	BIT	OP1 작업자 전등 ON Pb
P01516	BIT	W400 서보모터 도그3
M16977	BIT	OP1 수동용접기 Power On Lamp
D139240	WORD	PLC -> PC 실시간 DATA W480 1차스캔 품번
D139246	WORD	PLC -> PC 실시간 DATA W480 1차스캔 ALC코드
D139250	WORD	PLC -> PC 실시간 DATA W480 1차스캔 생산 년,월,일
D139253	WORD	PLC -> PC 실시간 DATA W480 1차스캔 생산카운터
D139260	WORD	PLC -> PC 실시간 DATA W480 2차스캔 품번
D139266	WORD	PLC -> PC 실시간 DATA W480 2차스캔 ALC코드
D139270	WORD	PLC -> PC 실시간 DATA W480 2차스캔 생산 년,월,일
D139273	WORD	PLC -> PC 실시간 DATA W480 2차스캔 생산카운터
D120200	WORD	PLC -> PC W130 1차스캔 DATA
D120220	WORD	PLC -> PC W130 2차스캔 DATA
D120000	WORD	W130 스캔 DATA
D121000	WORD	W100 DATA
D102001	WORD	PLC -> PC 반입 카운터
D102009	WORD	PLC -> PC 정상 투입여부
M01626	BIT	W150-2 파트체크 정상
M01627	BIT	W150-2 차종감지 파트정상
M0162F	BIT	W150-2 차광막 하강/상승
M01630	BIT	W150-2 양수기동 이상
M01631	BIT	W150-2 Anti-Repeat
M01632	BIT	W150-2 기동 Pulse
M01641	BIT	W150-2 로딩 로보트 간섭무
M01642	BIT	W150-2 언로딩 로보트 간섭무
M01643	BIT	W150-2 Work Robot 간섭무
M01670	BIT	W150-2 기동준비
M01671	BIT	W150-2 1차 기동
M01672	BIT	W150-2 2차 기동
M01673	BIT	W150-2 3차 기동
M01674	BIT	W150-2 4차 기동
M01679	BIT	W150-2 1차 작업준비
M0167A	BIT	W150-2 2차 작업준비
M01681	BIT	W150-2 1차 기동 End
M01682	BIT	W150-2 2차 기동 End
M01683	BIT	W150-2 3차 기동 End
T1603	BIT/WORD	W150-2 Air Blow On TMR
T1612	BIT/WORD	W150-2 로보트 간섭무지연
T1616	BIT/WORD	W150-2 파트이상 (누락)지연
T1630	BIT/WORD	W150-2 양수기동 이상지연